PROGRAM AnalogSignals

analogSignals_ex07();

END_PROGRAM

(* stored: Version 1.1.0.1
   POU AnalogSignals: Id {9204c07b-a1f6-4457-b29f-f2f8200423b3}, SpecialFunc None *)
